// TIA Portal V16 export
// export: Created 2022-03-06T01:43:08.9915725Z, ExportSetting WithDefaults, DisplayName Totally Integrated Automation Portal, DisplayVersion V16 Update 4, DisplayName TIA Portal Version Control Interface, DisplayVersion V16 Update 2, DisplayName TIA Portal Openness, DisplayVersion V16 Update 4, DisplayName TIA Portal Teamcenter Gateway, DisplayVersion V16, DisplayName SINAMICS Startdrive Advanced, DisplayVersion V16 Update 4, DisplayName SINAMICS Startdrive G110M, G120, G120C, G120D, G120P, G115D, DisplayVersion V16 Update 4, DisplayName SINAMICS Startdrive G130, G150, S120, S150, SINAMICS MV, S210, DisplayVersion V16 Update 4, DisplayName STEP 7 Professional, DisplayVersion V16 Update 4, DisplayName STEP 7 Safety, DisplayVersion V16, DisplayName WinCC Advanced / Unified PC, DisplayVersion V16 Update 4
FUNCTION "Escalamiento_G120" : Void   // FC10, LAD
{ S7_Optimized_Access := 'TRUE' }
VERSION : 0.1
// stored: AutoNumber false, IsIECCheckEnabled false, SetENOAutomatically false, UDAEnableTagReadback false
   VAR_TEMP
      vactual_norm : Real;
      setpoint_norm : Real;
   END_VAR
BEGIN

REGION Network 1: Escalar Velocidad actual
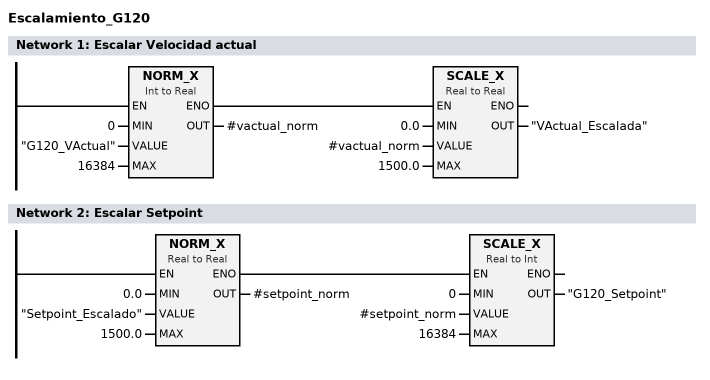
   RUNG wire#powerrail
      { S7_Templates := "[SrcType := Int, DestType := Real]" } Normalize(min := 0, value := "G120_VActual", max := 16384, out => #vactual_norm)
      { S7_Templates := "[SrcType := Real, DestType := Real]" } Scale(min := 0.0, value := #vactual_norm, max := 1500.0, out => "VActual_Escalada")
   END_RUNG
   // the same network as SCL:
   #vactual_norm := NORM_X(MIN := 0, VALUE := "G120_VActual", MAX := 16384);
   "VActual_Escalada" := SCALE_X(MIN := 0.0, VALUE := #vactual_norm, MAX := 1500.0);
END_REGION

REGION Network 2: Escalar Setpoint
   RUNG wire#powerrail
      { S7_Templates := "[SrcType := Real, DestType := Real]" } Normalize(min := 0.0, value := "Setpoint_Escalado", max := 1500.0, out => #setpoint_norm)
      { S7_Templates := "[SrcType := Real, DestType := Int]" } Scale(min := 0, value := #setpoint_norm, max := 16384, out => "G120_Setpoint")
   END_RUNG
   // the same network as SCL:
   #setpoint_norm := NORM_X(MIN := 0.0, VALUE := "Setpoint_Escalado", MAX := 1500.0);
   "G120_Setpoint" := SCALE_X(MIN := 0, VALUE := #setpoint_norm, MAX := 16384);
END_REGION
END_FUNCTION
